FUNCTION Robot2World 
VAR_INPUT
	vx_robot: 	 LREAL;
	vy_robot: 	 LREAL;
	omega_robot: LREAL;
	theta: 		 LREAL;
END_VAR

VAR_OUTPUT
	vx_world: 	 LREAL;
	vy_world: 	 LREAL;
	omega_world: LREAL;
END_VAR

VAR
END_VAR

vx_world 	:= COS(theta)*vx_robot - SIN(theta)*vy_robot;
vy_world 	:= SIN(theta)*vx_robot + COS(theta)*vy_robot;
omega_world := omega_robot;

END_FUNCTION

(* stored: Version 1.1.0.1, ProductVersion 3.1.4024.11
   POU Robot2World: Id {43a0fc94-b010-4129-bae3-4a831e83fafa}, SpecialFunc None *)
